FUNCTION Array2D_Cols : UINT
VAR_IN_OUT CONSTANT
	A : ARRAY[*,*] OF LREAL;
END_VAR

IF UPPER_BOUND(A,2) < LOWER_BOUND(A,2) THEN
	Array2D_Cols := 0;
ELSE
	Array2D_Cols := DINT_TO_UINT(UPPER_BOUND(A,2) - LOWER_BOUND(A,2) + 1);
END_IF

END_FUNCTION

(* stored: Version 1.1.0.1, ProductVersion 3.1.4024.9
   POU Array2D_Cols: Id {d9bcbe95-24ed-0e70-18e9-d3b65c6ff74f}, SpecialFunc None *)
